(* CoDeSys 2.3.9.41 project: WASCHSTRASSE.pro *)
(* Libraries: STANDARD.LIB 5.6.98 11:03:02 *)

(* Task configuration *)
TASK Standard (PRIORITY := 0, INTERVAL := T#1ms);
	MAIN
END_TASK

(* Global variable list: Global_Variables *)
VAR_GLOBAL
	(* Input *)
	S1 AT %I* : BOOL;
	S2 AT %I* : BOOL;
	I AT %I* : BOOL;
	L1 AT %I* : BOOL;
	L2 AT %I* : BOOL;
	L3 AT %I* : BOOL;
	(* Output *)
	RED AT %Q* : BOOL;
	GREEN AT %Q* : BOOL;
	K1 AT %Q* : BOOL;
	K2 AT %Q* : BOOL;
	K3 AT %Q* : BOOL;
	K4 AT %Q* : BOOL;
END_VAR
VAR_GLOBAL CONSTANT
	T : UINT := 1;
END_VAR

(* Data type *)
TYPE st_fsm_t :
(
	ST_OFF := 1,
	ST_ON,
	ST_WAIT,
	ST_START,
	ST_L1,
	ST_L2
);
END_TYPE

(* POU MAIN, ST *)
PROGRAM MAIN
VAR
	WASCHSTRASSE : FSM;
END_VAR
WASCHSTRASSE();
END_PROGRAM

(* POU FSM, ST *)
FUNCTION_BLOCK FSM
VAR_INPUT
END_VAR
VAR_OUTPUT
END_VAR
VAR
	state : st_fsm_t := ST_OFF;
	cnt : UINT := 2000;
END_VAR
CASE state OF
ST_OFF:
	IF S2 = TRUE THEN
		state := ST_ON;
	END_IF
ST_ON:
	GREEN := 1;
	RED := 0;
	K1 := 0;
	K2 := 0;
	K3 := 0;
	K4 := 0;
	IF S1 = 1 AND I = 1 AND K1 = 0 AND K2 = 0 AND K3 = 0 AND K4 = 0 THEN
		state := ST_WAIT;
		cnt := 2000;
	END_IF
ST_WAIT:
	IF cnt >= 0 THEN
		cnt := cnt - T;
	ELSE
		state := ST_START;
	END_IF
ST_START:
	K1 := 1;
	IF L1 = 1 THEN
		state := ST_L1;
	END_IF
ST_L1:
	K2 := 1;
	K3 := 1;
	GREEN := 0;
	RED := 1;
	IF L2 = 1 THEN
		state := ST_L2;
	END_IF	;
ST_L2:
	K2 := 0;
	K3 := 0;
	K4 := 1;
	IF L3 = 1 THEN
		state := ST_ON;
	END_IF	;
ELSE
	state := ST_OFF;
END_CASE
END_FUNCTION_BLOCK
